// TwinCAT 3 PLC project Sample01
// ProgramVersion: 3.1.4020.1
// libraries:
//   Tc2_Standard, * (Beckhoff Automation GmbH)
//   Tc2_System, * (Beckhoff Automation GmbH)
//   Tc3_Module, * (Beckhoff Automation GmbH)
// project tree:
//   / PlcTask.TcTTO
//   POUs/ F_CalcSum1DimArrayOldSchool.TcPOU, MAIN.TcPOU
// real-time tasks:
//   TASK PlcTask: cycle T#10ms, priority 20, ADS port 350

CONFIGURATION Sample01
    RESOURCE PLC ON TwinCAT3
        TASK PlcTask(INTERVAL := T#10ms, PRIORITY := 20);
        PROGRAM MAIN WITH PlcTask : MAIN;
    END_RESOURCE
END_CONFIGURATION

// ---- POUs/MAIN.TcPOU
PROGRAM MAIN
VAR
	array01 	: ARRAY[2..8] OF LREAL := [16.1, 34.1, 4.1, 43.1, 35.1, 2.1, 65.1];
	lrSum01		: LREAL;
	
	array02		: ARRAY[-1..2] OF LREAL := [16.1, 34.1, 9.1, 13.1];
	lrSum02		: LREAL;
	
	array03 	: ARRAY[-3..-1] OF LREAL := [16.1, 34.1, 8.1];
	lrSum03		: LREAL;
END_VAR

lrSum01 := F_CalcSum1DimArrayOldSchool(ADR(array01), SIZEOF(array01));
lrSum02 := F_CalcSum1DimArrayOldSchool(ADR(array02), SIZEOF(array02));
lrSum03 := F_CalcSum1DimArrayOldSchool(ADR(array03), SIZEOF(array03));

END_PROGRAM

// ---- POUs/F_CalcSum1DimArrayOldSchool.TcPOU
FUNCTION F_CalcSum1DimArrayOldSchool : LREAL
VAR_INPUT
	pData			: POINTER TO LREAL;
	nSize			: UDINT;
END_VAR
VAR
	pDataIndex		: POINTER TO LREAL;
	nUpperIndex		: UDINT;
	nIndex			: UDINT;
END_VAR

F_CalcSum1DimArrayOldSchool := 0;
nUpperIndex := nSize / SIZEOF(pDataIndex^);
IF (nUpperIndex > 0) THEN
	FOR nIndex := 0 TO (nUpperIndex - 1) DO
		pDataIndex := pData + (nIndex * SIZEOF(pDataIndex^));
		F_CalcSum1DimArrayOldSchool := F_CalcSum1DimArrayOldSchool + pDataIndex^;	
	END_FOR
END_IF

END_FUNCTION
